{region '#Template'}
	{attribute 'Version' := '5.0.0.0'}
	{attribute 'Tags' := '"LCID": "1031", "Text": "GVL, Allgemein, Notification classes, Event classes ID"'}
	{attribute 'Tags' := '"LCID": "1033", "Text": "GVL, General, Notification classes, Event classes ID"'}
	{attribute 'Description' := '"LCID": "1031", "Text": "Ereignisklassen"'}
	{attribute 'Description' := '"LCID": "1033", "Text": "Event classes"'}
{endregion}

{attribute 'qualified_only'}
VAR_GLOBAL CONSTANT
	NC10							: UDINT := 10; // Gefahr für Leben // Danger to life	
	NC20							: UDINT := 20; // Sicherheitsmeldung // Safety message	
	NC30							: UDINT := 30; // Alarmeldung // Alarm message	
	NC40							: UDINT := 40; // Störungsmeldung // Fault message	
	NC50							: UDINT := 50; // Wartungsmeldung // Maintenance message	
	NC51							: UDINT := 51; // Wartungsmeldung // Maintenance message	
	NC60							: UDINT := 60; // Systemmeldung // System message	
	NC70							: UDINT := 70; // Handeingriff // Manual operation	
	NC80							: UDINT := 80; // Sonstige Meldungen // Other message	
END_VAR

(* stored: Version 1.1.0.1, ProductVersion 3.1.4024.12
   GVL EC_ID: Id {358e0f7e-9d30-4f2e-9eba-e43d70ec62c1} *)
